PROGRAM prg_Opslagvat
VAR
	SensorHoog		AT		%I*		:BOOL;
	SensorLaag		AT		%I*		:BOOL;
	StartKnop		AT		%I*		:BOOL;
	StopKnop		AT		%I*		:BOOL;
	
	Klep			AT		%Q*		:BOOL;
	Pomp			AT		%Q*		:BOOL;
	Vullen			AT		%Q*		:BOOL;
END_VAR

Klep := SensorLaag AND NOT(SensorHoog);
Vullen := SensorLaag AND NOT(SensorHoog);

IF StopKnop OR SensorLaag THEN
	Pomp := FALSE;
ELSIF StartKnop AND NOT Vullen THEN
	Pomp := TRUE; 
END_IF

END_PROGRAM

(* stored: Version 1.1.0.1, ProductVersion 3.1.4024.15
   POU prg_Opslagvat: Id {a9d293a4-d2f4-4668-a4b2-c79a3cbb2abb}, SpecialFunc None *)
